(*********************************** G.D S.p.A. - Technical Department ***********************************
============= PROGRAM INFO ============
FOLDER:             TBD
MACHINES INVOLVED:  TBD 

============= DESCRIPTION =============
WU phase manager snapshot set function

============= REVISIONS ===============
Date		Version	 	Author      	Description             
----------	-------		------------  	--------------------------------------------
2020/06/19 	0000.00	 	G.Cera 			Creation of the PRG

**********************************************************************************************************)

FUNCTION csp_main_phaseManager_set_snapshot : VOID
VAR_INPUT
    errorID_1:				DINT;			(* Field for specify the faults code or enter
								   				more message info *)
    errorID_2:				DINT;			(* Field for specify the faults code or enter
								   				more message info *)
    errorID_3:				DINT;			(* Field for specify the faults code or enter
								   				more message info *)
	reason:					STRING := '';

	job_not_scheduled:		BOOL;
	
	job_pending:			BOOL;
	
END_VAR

VAR_IN_OUT
    CONVERSION_this:		csp_main_phaseManager_snapshot;
								(* csp_main_phaseManager_snapshot snapshot reference *)
END_VAR

IF	message_set(
		errorID_1		:= errorID_1, 
		errorID_2		:= errorID_2, 
		errorID_3		:= errorID_3, 
		CONVERSION_this	:= CONVERSION_this.message)
THEN
	CONVERSION_this.reason 				:= reason;
	CONVERSION_this.job_not_scheduled	:= job_not_scheduled;
	CONVERSION_this.job_pending			:= job_pending;
END_IF

END_FUNCTION

(* stored: Version 1.1.0.1, ProductVersion 3.1.4024.3
   POU csp_main_phaseManager_set_snapshot: Id {4694ae41-7e92-0b70-2adc-f74ae464682c}, SpecialFunc None *)
